(* IEC 61131-3 sources: AXOpen/src/components.kuka.robotics/app/src/Documentation, 3 files *)

(* ---- Component_1.st ---- *)
USING AXOpen.Core;

NAMESPACE AXOpen.Components.Kuka.Robotics
    {S7.extern=ReadWrite}
    CLASS Component_1 EXTENDS AXOpen.Core.AxoObject
        //<ComponentDeclaration>
        VAR PUBLIC
            ExampleRobot : AXOpen.Components.Kuka.Robotics.AxoKrc4_v_5_x_x;
        END_VAR
        //</ComponentDeclaration>

        //<InitializationArgumentsDeclaration>
        VAR PUBLIC
            movementParams : AXOpen.Components.Abstractions.Robotics.AxoRoboticsMovementsParams;
            {#ix-set:AttributeName = "<#Activate manual control#>"}
            ActivateManualControl : BOOL;
        END_VAR
        //</InitializationArgumentsDeclaration>

        METHOD PUBLIC Run
            VAR_INPUT
                parent : IAxoContext;
            END_VAR

            THIS.Initialize(parent);

            IF ActivateManualControl THEN
                ExampleRobot.ActivateManualControl();
            END_IF;

            //<Initialization>
            ExampleRobot.Run(THIS,
                                HwIdentifiers#KRC4_HwID,
                                HwIdentifiers#KRC4_512_digital_in_and_outputs_1_512_digital_in__and_outputs_HwID);
            //</Initialization>

        THIS.UseInSequencer();
        END_METHOD

        //<Usage>
        VAR PUBLIC
            Sequencer : AxoSequencer;
            Steps : ARRAY[0..3] OF AXOpen.Core.AxoStep;
        END_VAR

        METHOD PRIVATE UseInSequencer

            Sequencer.Initialize(THIS);
            Sequencer.Open();

            IF(Steps[0].Execute(Sequencer, 'Start at main')) THEN
                IF(ExampleRobot.StartAtMain().IsDone()) THEN
                    Sequencer.MoveNext();
                END_IF;
            END_IF;

            IF(Steps[1].Execute(Sequencer, 'Move to position')) THEN
                IF(ExampleRobot.StartMovements(movementParams).IsDone()) THEN
                    Sequencer.MoveNext();
                END_IF;
            END_IF;

            IF(Steps[1].Execute(Sequencer, 'Stop')) THEN
                IF(ExampleRobot.StopMovements().IsDone()) THEN
                    Sequencer.CompleteSequence();
                END_IF;
            END_IF;
        END_METHOD

        //</Usage>
    END_CLASS
END_NAMESPACE

(* ---- Component_2.st ---- *)
USING AXOpen.Core;

NAMESPACE AXOpen.Components.Kuka.Robotics
    {S7.extern=ReadWrite}
    CLASS Component_2 EXTENDS AXOpen.Core.AxoObject
        //<ComponentDeclaration>
        VAR PUBLIC
            ExampleRobot : AXOpen.Components.Kuka.Robotics.AxoKrc4_v_5_x_x;
        END_VAR
        //</ComponentDeclaration>

        //<InitializationArgumentsDeclaration>
        VAR PUBLIC
            movementParams : AXOpen.Components.Abstractions.Robotics.AxoRoboticsMovementsParams;
            {#ix-set:AttributeName = "<#Activate manual control#>"}
            ActivateManualControl : BOOL;
        END_VAR
        //</InitializationArgumentsDeclaration>

        METHOD PUBLIC Run
            VAR_INPUT
                parent : IAxoContext;
            END_VAR

            THIS.Initialize(parent);

            IF ActivateManualControl THEN
                ExampleRobot.ActivateManualControl();
            END_IF;

            //<Initialization>
            ExampleRobot.Run(THIS,
                                HwIdentifiers#KRC4_HwID,
                                HwIdentifiers#KRC4_512_digital_in_and_outputs_1_512_digital_in__and_outputs_HwID);
            //</Initialization>

        THIS.UseInSequencer();
        END_METHOD

        //<Usage>
        VAR PUBLIC
            Sequencer : AxoSequencer;
            Steps : ARRAY[0..3] OF AXOpen.Core.AxoStep;
        END_VAR

        METHOD PRIVATE UseInSequencer

            Sequencer.Initialize(THIS);
            Sequencer.Open();

            IF(Steps[0].Execute(Sequencer, 'Start at main')) THEN
                IF(ExampleRobot.StartAtMain().IsDone()) THEN
                    Sequencer.MoveNext();
                END_IF;
            END_IF;

            IF(Steps[1].Execute(Sequencer, 'Move to position')) THEN
                IF(ExampleRobot.StartMovements(movementParams).IsDone()) THEN
                    Sequencer.MoveNext();
                END_IF;
            END_IF;

            IF(Steps[1].Execute(Sequencer, 'Stop')) THEN
                IF(ExampleRobot.StopMovements().IsDone()) THEN
                    Sequencer.CompleteSequence();
                END_IF;
            END_IF;
        END_METHOD

        //</Usage>
    END_CLASS
END_NAMESPACE

(* ---- DocumentationContext.st ---- *)
NAMESPACE AXOpen.Components.Kuka.Robotics
    {S7.extern=ReadWrite}
    CLASS DocumentationContext EXTENDS AXOpen.Core.AxoContext
        VAR PUBLIC
            _rootObject : AxoObject;
            componentOne : Component_1;
            componentTwo : Component_2;
        END_VAR

        METHOD PROTECTED OVERRIDE Main
            THIS.InitializeRootObject(_rootObject);
            componentOne.Run(_rootObject);
            RETURN;
            componentTwo.Run(_rootObject);
        END_METHOD
    END_CLASS
END_NAMESPACE
